FUNCTION_BLOCK Train1
  (* Standard: 61499-2 *)
  (* Version 0.1, 2017-00-23, hpea485, UOA *)
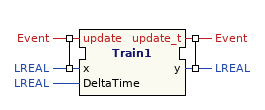
  EVENT_INPUT
    update WITH x;
  END_EVENT
  EVENT_OUTPUT
    update_t WITH y;
  END_EVENT
  VAR_INPUT
    x : LREAL;
    DeltaTime : LREAL := 1;
  END_VAR
  VAR_OUTPUT
    y : LREAL;
  END_VAR
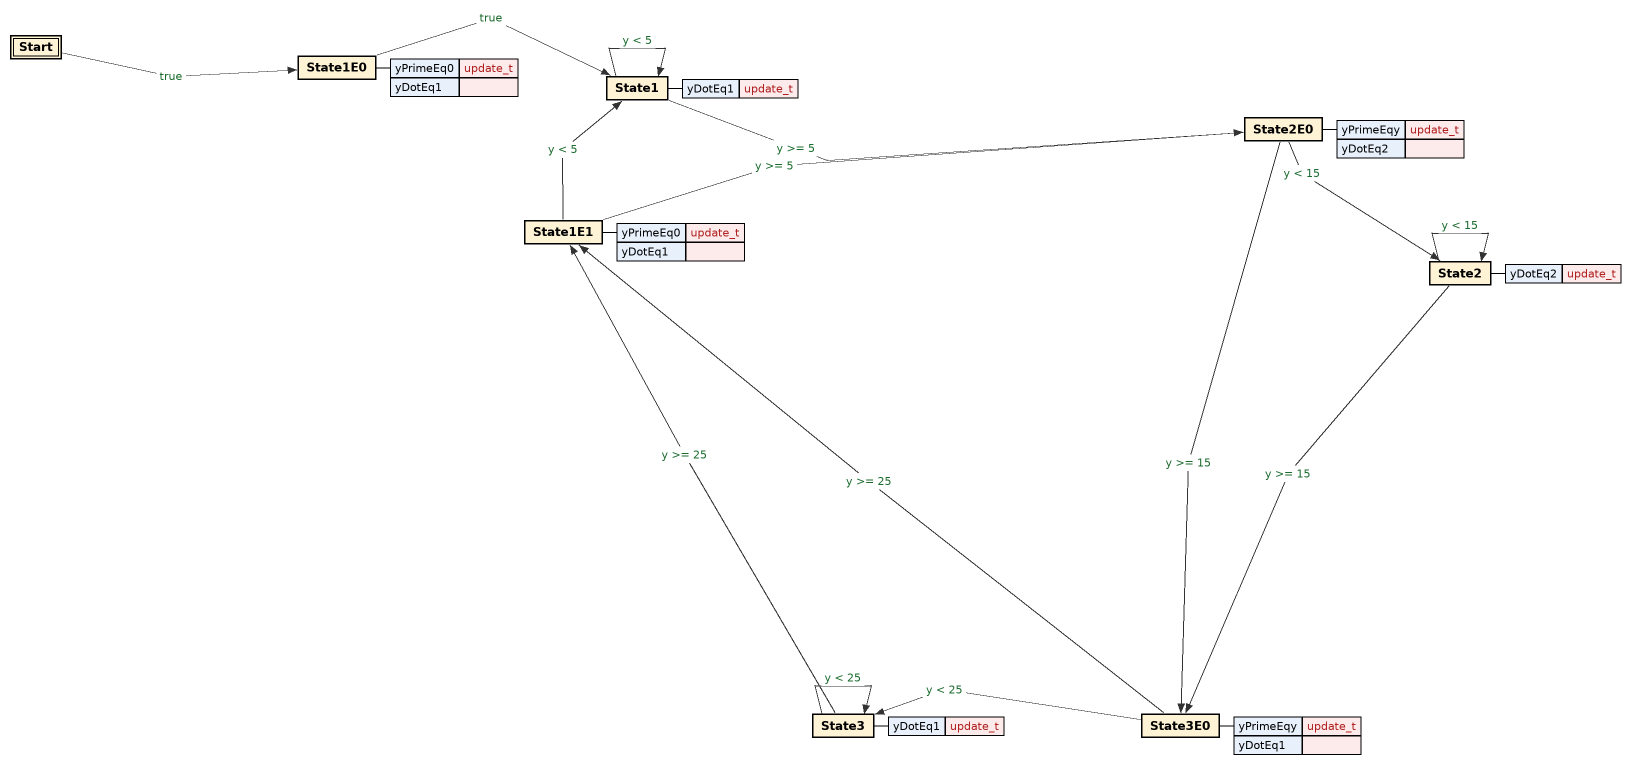
  EC_STATES
    Start;
    State1E0 : yPrimeEq0 -> update_t, yDotEq1;
    State1 : yDotEq1 -> update_t;
    State2E0 : yPrimeEqy -> update_t, yDotEq2;
    State2 : yDotEq2 -> update_t;
    State3E0 : yPrimeEqy -> update_t, yDotEq1;
    State3 : yDotEq1 -> update_t;
    State1E1 : yPrimeEq0 -> update_t, yDotEq1;
  END_STATES
  EC_TRANSITIONS
    Start TO State1E0 := true;
    State1E0 TO State1 := true;
    State1 TO State2E0 := y >= 5;
    State1 TO State1 := y < 5;
    State2E0 TO State2 := y < 15;
    State2E0 TO State3E0 := y >= 15;
    State2 TO State3E0 := y >= 15;
    State2 TO State2 := y < 15;
    State3E0 TO State3 := y < 25;
    State3E0 TO State1E1 := y >= 25;
    State3 TO State1E1 := y >= 25;
    State3 TO State3 := y < 25;
    State1E1 TO State1 := y < 5;
    State1E1 TO State2E0 := y >= 5;
  END_TRANSITIONS
  ALGORITHM yDotEq1 IN C: (* ODE *)
y_dot = 1;
  END_ALGORITHM
  ALGORITHM yDotEq2 IN C: (* ODE *)
y_dot = 2;
  END_ALGORITHM
  ALGORITHM yPrimeEq0 IN C: (* ODE_init *)
y_prime = 0;
  END_ALGORITHM
  ALGORITHM yPrimeEqy IN C: (* ODE_init *)
y_prime = y;
  END_ALGORITHM
END_FUNCTION_BLOCK
